(* CODESYS project control1 -v2.export

Project tree, tasks and I/O mapping:
  CODESYS_Control_Win_V3_x64 : CODESYS Control Win V3 x64, 3S - Smart Software Solutions GmbH, version 3.5.16.0
    application Application
      libraries: Standard, * (System); CAA Tick Extern, 3.5.7.0 (CAA Technical Workgroup); MQTT, 1.1.0.2 (Stefan Dreyer); Common Helper for development, 1.0.0.0 (Stefan Dreyer)
      task Task (freewheeling, priority 1) calls MQTT_Prog, LogicControl
      task VISU_TASK (cyclic, interval 100 ms, priority 31) calls VisuElems.Visu_Prg
      global variables GVL
      program LogicControl [CFC]
      program MQTT_Prog [ST]
      function block StringReceiver [ST]: PublishReceived
      visualisation Visualization
  libraries: VisuSymbols, 3.5.10.0 (System)
  text list GlobalTextList
*)

// CODESYS_Control_Win_V3_x64/Application/GVL
{attribute 'qualified_only'}
VAR_GLOBAL
	count: WORD := 0;
	u1 : BOOL;
	u2 : BOOL;
	y2 : BOOL;
	s1 : BOOL;
	s2 : BOOL;
END_VAR

// CODESYS_Control_Win_V3_x64/Application/MQTT_Prog
PROGRAM MQTT_Prog
VAR
	//first reciver for MQTT String
	stringu1 : StringReceiver;
	strings2 : StringReceiver;
	
	//the collector
	Collector:SD_MQTT.CallbackCollector;
	//the client
	Client:SD_MQTT.HANDLE_MQTT;
	MQTT_IN_OUT:SD_MQTT.MQTT_IN_OUT;
	//your special client id
	ClientID:STRING;
	S1 : STRING;
	S2 : STRING;
	
	stateu1 : SD_MQTT.MQTTState;
	states2 : SD_MQTT.MQTTState;
	
	subscriber:SD_MQTT.MQTTSubscribe;
	
	init: BOOL;
	i:UINT;
	t1:ton;
	t2:ton;
END_VAR

S1 := CONCAT('stringu1:',TO_STRING(GVL.u1));
S2 := CONCAT('strings2:',TO_STRING(GVL.s2));

IF NOT init THEN
	init := TRUE;
	//collect all callbacks...
	
	Collector.put(stringu1);
	Collector.put(strings2);
	
	ClientID := CONCAT('CodesysMqtt',TO_STRING(TICKS.GetTick(xDummy:= TRUE)));
	MQTT_IN_OUT.ClientID := ClientID;
	subscriber.SetMqttInOut(MQTT_IN_OUT:= ADR(MQTT_IN_OUT));

	(*Target String1()*)
	stateu1.Init(
	State:= ADR(t1.Q), 
	Topic:= ADR('Codesys/Control/Vars'), (*here place the name of you instance*) 
	StateValueOn:= ADR(S1), 
	StateValueOff:= ADR(S1), 
	MQTT_IN_OUT:= ADR(MQTT_IN_OUT), 
	QoS:= SD_MQTT.QoS.ExactlyOnce,
	RetainMqtt:= FALSE,
	StateName:= ADR(''));
	
	states2.Init(
	State:= ADR(t1.Q), 
	Topic:= ADR('Codesys/Control/Vars'), (*here place the name of you instance*) 
	StateValueOn:= ADR(S2), 
	StateValueOff:= ADR(S2), 
	MQTT_IN_OUT:= ADR(MQTT_IN_OUT), 
	QoS:= SD_MQTT.QoS.ExactlyOnce,
	RetainMqtt:= FALSE,
	StateName:= ADR(''));
END_IF

Client(
	MQTT_IN_OUT:= MQTT_IN_OUT, 
	ENABLE:= TRUE, 
	URL:= 'test.mosquitto.org', 
	TIMEOUT:= T#5S);

	
subscriber(
	Subscribe:= TRUE, 
	Topic:= ADR('Codesys/Control/Vars'), 
	QoSSubscribe:= SD_MQTT.QoS.ExactlyOnce, 
	ExpectingString:= TRUE, 
	Callback:= Collector,
	);
//make a clock pulse...
t1(IN := NOT t2.Q, PT:= T#2S);
t2(IN := t1.Q, PT:= T#2S);

stateu1();  //publish
states2();

stringu1();  //subscribe
GVL.u2 := STRING_TO_BOOL(stringu1.MQTTString.MQTTReceived);
strings2();
GVL.s1 := STRING_TO_BOOL(strings2.MQTTString.MQTTReceived);

END_PROGRAM

// CODESYS_Control_Win_V3_x64/Application/StringReceiver
//this is needed for FBinstance name in Variable
{attribute 'reflection'}
FUNCTION_BLOCK StringReceiver IMPLEMENTS SD_MQTT.MQTT_SUBSCRIBE_CALLBACK
VAR_INPUT
END_VAR
VAR_OUTPUT
END_VAR
VAR
	//from this instance i can get my string...
	MQTTString:SD_MQTT.ReceiveString;
	init: BOOL;
	{attribute 'instance-path'}
	{attribute 'noinit'}
	instanceName: STRING(255);//this string contains the instance name of the FB
	//here we get the "lowest" element of the name...
	LastTreeName:STRING;
	StringPointer:POINTER TO STRING;
END_VAR

IF NOT init THEN
	init := TRUE;
	StringPointer := CommonTypesAndFunctions.FindLastDot(ADR(instanceName));
	
	StringPointer := StringPointer + SIZEOF(BYTE);
	
	LastTreeName := StringPointer^; 
	MQTTString.initAsFindPayload(compString:=ADR(LastTreeName), returnHit:= TRUE, splitChar:= ':');
END_IF


METHOD PublishReceived : BOOL
VAR_INPUT
	(*Collection of recived Data*)
	Data	: SD_MQTT.CALLBACK_DATA;
END_VAR
PublishReceived := MQTTString.PublishReceived(Data:= Data);
END_METHOD

END_FUNCTION_BLOCK

// CODESYS_Control_Win_V3_x64/Application/LogicControl
PROGRAM LogicControl
VAR
	SWITCH: BOOL;
END_VAR

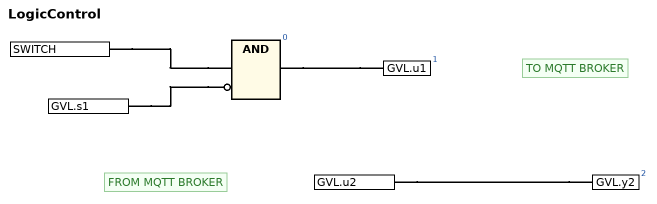
// TO MQTT BROKER
GVL.u1 := SWITCH AND NOT GVL.s1;
// FROM MQTT BROKER
GVL.y2 := GVL.u2;

END_PROGRAM

// CODESYS_Control_Win_V3_x64/Application/Visualization
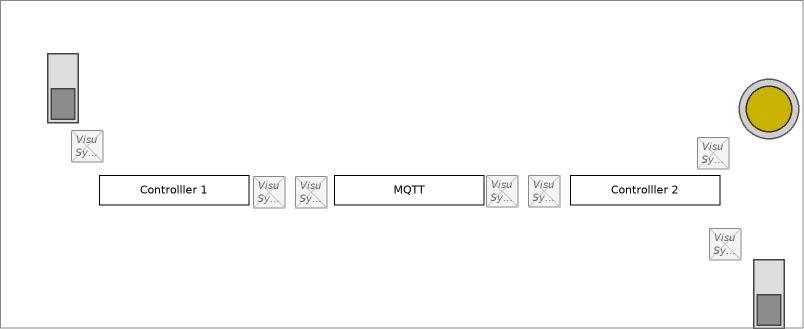
VISUALIZATION Visualization  // 804x329
    DipSwitch (28,53 70x70), variable: LogicControl.SWITCH, behaviour: TOGGLE, style: Switch-DipSwitch-Gray
    Lamp1 (734,74 70x70), variable: GVL.y2, style: Lamp-Lamp1-Yellow
    DipSwitch (734,259 70x70), variable: GVL.s2, behaviour: TOGGLE, style: Switch-DipSwitch-Gray
    Rectangle (334,175 150x30), "MQTT"
    Rectangle (99,175 150x30), "Controlller 1"
    Rectangle (570,175 150x30), "Controlller 2"
    Image (253,176 32x32), image: VisuSymbols.Symbols.ArrowBoldLeft
    Image (295,176 32x32), image: VisuSymbols.Symbols.ArrowBoldRight
    Image (486,175 32x32), image: VisuSymbols.Symbols.ArrowBoldLeft
    Image (528,175 32x32), image: VisuSymbols.Symbols.ArrowBoldRight
    Image (71,130 32x32), image: VisuSymbols.Symbols.ArrowBoldRightDown
    Image (697,137 32x32), image: VisuSymbols.Symbols.ArrowBoldRightUp
    Image (709,228 32x32), image: VisuSymbols.Symbols.ArrowBoldLeftUp
END_VISUALIZATION
